FUNCTION_BLOCK FOURTH_ORDER_SYSTEM (* 4rd ordem system *)
  (* Standard: 61499-2 *)
  (* Version 11-01-12, GASR *)
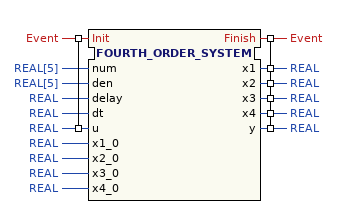
  EVENT_INPUT
    Init WITH u;
  END_EVENT
  EVENT_OUTPUT
    Finish WITH x1, x2, x3, x4, y;
  END_EVENT
  VAR_INPUT
    num : ARRAY [0..4] OF REAL;
    den : ARRAY [0..4] OF REAL;
    delay : REAL := 0;
    dt : REAL;
    u : REAL;
    x1_0 : REAL; (* initial condition *)
    x2_0 : REAL;
    x3_0 : REAL;
    x4_0 : REAL;
  END_VAR
  VAR_OUTPUT
    x1 : REAL;
    x2 : REAL;
    x3 : REAL;
    x4 : REAL;
    y : REAL;
  END_VAR
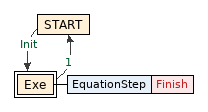
  EC_STATES
    Exe : EquationStep -> Finish;
    START;
  END_STATES
  EC_TRANSITIONS
    Exe TO START := 1;
    START TO Exe := Init;
  END_TRANSITIONS
  ALGORITHM EquationStep IN Lua: (* num[1] = b0, num[2] = b1 *)

						if type(input_buffer) ~= 'table' then
							input_buffer = {}
							for i = 1, math.ceil(delay/dt) +2 do
								input_buffer[#input_buffer +1] = 0
							end
						end

						input_buffer[#input_buffer] = u
						u = input_buffer[1]
						for i = 1, #input_buffer-1 do
							input_buffer[i] = input_buffer[i+1]
						end


						local beta1 = (num[2] - den[2]*num[1])
						local beta2 = num[3] - den[2]*beta1 - den[3]*num[1];
						local beta3 = num[4] - den[2]*beta2 - den[3]*beta1 - den[4]*num[1];
						local beta4 = num[5] - den[2]*beta3 - den[3]*beta2 -den[4]*beta1 - den[5]*num[1];

						local function f1(X1, X2,X3, X4, U)
							return X2 + beta1*U
						end

						local function f2(X1, X2, X3,X4, U)
							return X3 + beta2*U
						end

						local function f3(X1, X2, X3, X4, U)
							return X4 + beta3*U
						end

						local function f4(X1, X2, X3, X4, U)
							return (-den[5]*X1 - den[4]*X2 - den[3]*X3 -den[2]*X4 + beta4*U)
						end

						R11 = dt*f1(x1_0, x2_0, x3_0, x4_0, u);
						R12 = dt*f2(x1_0, x2_0, x3_0, x4_0, u);
						R13 = dt*f3(x1_0, x2_0, x3_0, x4_0, u);
						R14 = dt*f4(x1_0, x2_0, x3_0, x4_0, u);

						x1aux = x1_0 + 0.5*R11
						x2aux = x2_0 + 0.5*R12
						x3aux = x3_0 + 0.5*R13
						x4aux = x4_0 + 0.5*R14



						R21 = dt*f1(x1aux, x2aux, x3aux, x4aux, u);
						R22 = dt*f2(x1aux, x2aux, x3aux, x4aux, u);
						R23 = dt*f3(x1aux, x2aux, x3aux, x4aux, u);
						R24 = dt*f4(x1aux, x2aux, x3aux, x4aux, u);

						x1aux = x1aux + 0.5*R21
						x2aux = x2aux + 0.5*R22
						x3aux = x3aux + 0.5*R23
						x4aux = x4aux + 0.5*R24

						R31 = dt*f1(x1aux, x2aux, x3aux, x4aux, u);
						R32 = dt*f2(x1aux, x2aux, x3aux, x4aux, u);
						R33 = dt*f3(x1aux, x2aux, x3aux, x4aux, u);
						R34 = dt*f4(x1aux, x2aux, x3aux, x4aux, u);

						x1aux = x1aux + 0.5*R31
						x2aux = x2aux + 0.5*R32
						x3aux = x3aux + 0.5*R33
						x4aux = x4aux + 0.5*R34

						R41 = dt*f1(x1aux, x2aux, x3aux, x4aux, u);
						R42 = dt*f2(x1aux, x2aux, x3aux, x4aux, u);
						R43 = dt*f3(x1aux, x2aux, x3aux, x4aux, u);
						R44 = dt*f4(x1aux, x2aux, x3aux, x4aux, u);


						x1 = x1_0 + (1/6)*(R11 + 2*R21 + 2*R31 + R41)
						x2 = x2_0 + (1/6)*(R12 + 2*R22 + 2*R32 + R42)
						x3 = x3_0 + (1/6)*(R13 + 2*R23 + 2*R33 + R43)
						x4 = x4_0 + (1/6)*(R14 + 2*R24 + 2*R34 + R44)


						y  = x1 + num[1]*u

						x1_0 = x1
						x2_0 = x2
						x3_0 = x3
						x4_0 = x4
  END_ALGORITHM
END_FUNCTION_BLOCK
(* other elements stored in the file *)
(* VarDeclaration Name=R11 Type=REAL *)
(* VarDeclaration Name=R12 Type=REAL *)
(* VarDeclaration Name=R13 Type=REAL *)
(* VarDeclaration Name=R14 Type=REAL *)
(* VarDeclaration Name=R21 Type=REAL *)
(* VarDeclaration Name=R22 Type=REAL *)
(* VarDeclaration Name=R23 Type=REAL *)
(* VarDeclaration Name=R24 Type=REAL *)
(* VarDeclaration Name=R31 Type=REAL *)
(* VarDeclaration Name=R32 Type=REAL *)
(* VarDeclaration Name=R33 Type=REAL *)
(* VarDeclaration Name=R34 Type=REAL *)
(* VarDeclaration Name=R41 Type=REAL *)
(* VarDeclaration Name=R42 Type=REAL *)
(* VarDeclaration Name=R43 Type=REAL *)
(* VarDeclaration Name=R44 Type=REAL *)
(* VarDeclaration Name=x1aux Type=REAL *)
(* VarDeclaration Name=x2aux Type=REAL *)
(* VarDeclaration Name=x3aux Type=REAL *)
(* VarDeclaration Name=x4aux Type=REAL *)
(* VarDeclaration Name=input_buffer Type=REAL *)
